# EPICS substitutions: tests/inputs/example_sub.substitutions
file db_with_readbacks.db
{
pattern {}
{}
}

file simple_db.db
{
pattern {}
{}
{}
{}
}
